// LS Electric XG5000 project: 12
// PLC LSPLC

PROGRAM NewProgram (task: 스캔 프로그램)

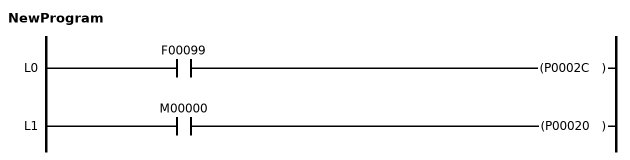
; L0
LOAD      F00099
OUT       P0002C
; L1
LOAD      M00000
OUT       P00020